// TIA Portal V16 export
// export: Created 2025-05-30T16:36:06.6173637Z, ExportSetting WithDefaults, DisplayName Totally Integrated Automation Portal, DisplayVersion V16, DisplayName TIA Portal Version Control Interface, DisplayVersion V16, DisplayName TIA Portal Openness, DisplayVersion V16, DisplayName STEP 7 Professional, DisplayVersion V16, DisplayName STEP 7 Safety, DisplayVersion V16, DisplayName WinCC Advanced, DisplayVersion V16
DATA_BLOCK "ProductBuffer_DB"   // DB58
VERSION : 0.1
// stored: AutoNumber true, InstanceOfName ProductBuffer, InstanceOfType FB
"ProductBuffer"
   // VAR_INPUT
   //    SensorInput : Bool;
   //    TimeDelay : Time;
   //    TriggerFeedback : Bool;
   // END_VAR
   // VAR_OUTPUT
   //    TriggerMovement : Bool;
   //    ProductCount : Int;
   // END_VAR
   // VAR RETAIN
   //    PrevSensor : Bool;
   //    DelayTimer : TON;
   //    MovementActive { S7_SetPoint := 'True'} : Bool;
   // END_VAR
BEGIN
END_DATA_BLOCK
